{attribute 'qualified_only'}
{attribute 'strict'}
TYPE PulsPisaChannelCount :
(
	FOUR := 4,
	EIGHT :=8
);
END_TYPE

(* stored: Version 1.1.0.1, ProductVersion 3.1.4024.15
   EnumerationTextList PulsPisaChannelCount: Id {0d17e9f4-3e22-418f-91ce-0f43fae7e71e} *)
